(* IEC 61131-3 sources: MotionTestBenchMaster/Logical/00_AID/Libraries/Sidel_Libraries/ITC/TCP_COM, 5 files *)

(* ---- TCP_COM.typ ---- *)
(********************************************************************
 * COPYRIGHT --
 ********************************************************************
 * Package: TCP
 * File: TCP.typ
 * Author: Marco.Nicoli
 * Created: October 25, 2016 : Initial version
 *********************************************************************)

TYPE
	TCP_DataType : 	STRUCT
		Connection_OK : BOOL;
		Com_Status : UINT; (*(0=Connect OK;1=Not Enabled;2=Error Sending;3=Error Receiving;10=Connection Waiting)*)
		Recv_Buffer : ARRAY[0..20]OF USINT;
		Send_Buffer : ARRAY[0..20]OF USINT;
	END_STRUCT;
	TCP_Status_Type :
		(
		DISABLED,
		INITIALIZE_FB,
		INITIAL_PING,
		READ_LOCAL_IP,
		OPEN_TCP,
		CFG_SERVER,
		CFG_CLIENT,
		ESTABLISHED_CONNECTION_AS_SERVER,
		ESTABLISHED_CONNECTION_AS_CLIENT,
		CLOSE1,
		CLOSE2,
		RECONNECTION
		);
	TCP_SendRec_Type :
		(
		COMM_IDLE,
		SEND_DATA,
		RECEIVE_DATA,
		COMM_PING
		);
	Ping_Status_Type :
		(
		NO_EXECUTION,
		EXECUTION,
		SUCCESSFUL,
		NO_RESPONSE,
		ERROR_INTERNAL
		);
END_TYPE

(* ---- PING_Fun.st ---- *)
FUNCTION_BLOCK PING_Fun
	IF NOT enable THEN
		PING_OK 			:= FALSE;
		ERR_NO_RESPONSE 	:= FALSE;
		ERR_INTERNAL	 	:= FALSE;
		ERROR 				:= FALSE;
		Status 				:= NO_EXECUTION;
		RETURN;
	END_IF;
	Fb_IcmpPing.pHost	:= ADR(IP_Address);
	Fb_IcmpPing.timeout := 50;
	CASE Status OF
		NO_EXECUTION:
			Fb_IcmpPing.enable  := FALSE;
			readResponse 	:= FALSE;
			PachetSent		:= 0;
			PachetRecived	:= 0;
			PachetLoss		:= 0;
			IF enable THEN
				Status := EXECUTION;
			END_IF;

		EXECUTION:
			Fb_IcmpPing.enable  := TRUE;
			IF Fb_IcmpPing.status = ERR_FUB_BUSY THEN
				readResponse := TRUE;
			END_IF
			IF readResponse THEN
				CASE Fb_IcmpPing.status OF
					ERR_OK:
						PachetSent 		:= PachetSent +1;
						PachetRecived 	:= PachetRecived +1;

					icmpERR_NO_RESPONSE:
						PachetSent 		:= PachetSent +1;
						PachetLoss 		:= PachetLoss +1;

					ERR_FUB_BUSY,
					ERR_FUB_ENABLE_FALSE:

					icmpERR_PARAMETER,
					icmpERR_SOCKET_CREATE,
					icmpERR_SYSTEM:
						Status := ERROR_INTERNAL;
				END_CASE;
			END_IF
			IF PachetSent >= 4 THEN
				IF PachetLoss >= 1 THEN
					Status := NO_RESPONSE;
				ELSE
					Status := SUCCESSFUL;
				END_IF
			END_IF

		SUCCESSFUL, NO_RESPONSE, ERROR_INTERNAL:
			Fb_IcmpPing.enable  := FALSE;

	END_CASE;
	Fb_IcmpPing();

	PING_OK 			:= Status = SUCCESSFUL;
	ERR_NO_RESPONSE 	:= Status = NO_RESPONSE;
	ERR_INTERNAL	 	:= Status = ERROR_INTERNAL;
	ERROR 				:= ERR_NO_RESPONSE OR ERR_INTERNAL;
END_FUNCTION_BLOCK

(* ---- TCP_COM.fun ---- *)
(********************************************************************
 * COPYRIGHT --
 ********************************************************************
 * Package: TCP
 * File: TCP.typ
 * Author: Marco.Nicoli
 * Created: October 25, 2016 : Initial version
 *********************************************************************)

FUNCTION_BLOCK TCP_COM (*TCP communication function*)
	VAR_INPUT
		Enable_Com : BOOL; (*Enable Communication*)
		Enable_Server : BOOL; (*Enable the server mode (False = Client mode | True = Serve mode)*)
		ETH_Card : STRING[16] := 'IF2'; (*Optional Parameter
Work with the following syntax when using IF2 on board:
IF2
Work with the following syntax when using a POWERLINK card:
SL<x>.SS<y>.IF<z>.PLKETH or SL<x>.SS<y>.IF<z>.ETH
*)
		IP_Address : STRING[16]; (*Partner IP address. (e.g. '10.1.92.20') (as a string)*)
		Local_Port : UINT; (*Local port number.*)
		Remote_Port : UINT; (*Remote port number.*)
		Recv_Buffer : UDINT; (*Received data buffer address (string given as a pointer)*)
		Recv_Length : UDINT; (*Reiceved data maximum length (in bytes)*)
		Send_Buffer : UDINT; (*Data to send buffer address (string given as a pointer)*)
		Send_Length : UDINT; (*Sent data length (in bytes)*)
		Send_Time_Act : TIME; (*Data send time cadence (in ms) (typical value: 100ms)*)
		Rcv_Time_Out : TIME; (*Reception time out setpoint (in ms) (typical value: 1000ms)*)
	END_VAR
	VAR_OUTPUT
		Connection_OK : BOOL; (*True = both PLCs are connected*)
		PING_OK : BOOL;
		ERROR : BOOL;
		ERR_NO_RESPONSE : BOOL;
		ERR_INTERNAL : BOOL;
	END_VAR
	VAR
		WhoIsConnected : STRING[16]; (*Connected client IP address*)
		IP_AdressLocal : STRING[16];
		TON_SendTime : TON;
		TON_RcvTimeOut : TON;
		TON_TCP_EnDelay : TON;
		TON_ConnectionTimeOut : TON;
		ConnectionAttempt : UINT;
		fb_Ping : PING_Fun;
		fb_TcpOpen : TcpOpen; (*Communication opening function block*)
		fb_TcpServer : TcpServer; (*Server creation function block*)
		fb_TcpClient : TcpClient; (*Client function block*)
		fb_TcpSend : TcpSend; (*Data sending function block*)
		fb_TcpRecv : TcpRecv; (*Data receiving function block*)
		fb_TcpClose : TcpClose; (*Communication closing function block*)
		fb_CfgGetIPAddr : CfgGetIPAddr;
		oldTCP_Status : TCP_Status_Type;
		oldTCP_CommStatus : TCP_SendRec_Type;
		IP_LocalValid : BOOL;
		readResponse : BOOL;
		commResponse : BOOL;
		TCP_Status : TCP_Status_Type; (*Implemented communication block status*)
		TCP_CommStatus : TCP_SendRec_Type; (*Implemented communication block status*)
		TON_Connection_OK : TON;
	END_VAR
END_FUNCTION_BLOCK

FUNCTION_BLOCK PING_Fun (*TODO: Add your comment here*) (*$GROUP=User,$CAT=User,$GROUPICON=User.png,$CATICON=User.png*)
	VAR_INPUT
		enable : BOOL;
		IP_Address : STRING[80];
	END_VAR
	VAR_OUTPUT
		PING_OK : BOOL;
		ERROR : BOOL;
		ERR_NO_RESPONSE : BOOL;
		ERR_INTERNAL : BOOL;
	END_VAR
	VAR
		Status : Ping_Status_Type;
		Fb_IcmpPing : IcmpPing;
		PachetRecived : USINT;
		PachetSent : USINT;
		PachetLoss : USINT;
		readResponse : BOOL;
	END_VAR
END_FUNCTION_BLOCK

(* ---- TCP_Fun.st ---- *)
(********************************************************************
 * COPYRIGHT --
 ********************************************************************
 * Package: TCP
 * File: TCP.st
 * Author: Marco.Nicolì
 * Created: October 25, 2016 : Initial version
 * Modified: November 15, 2016 : Something
 ********************************************************************)

FUNCTION_BLOCK TCP_COM
	CASE TCP_Status OF
		DISABLED:
			ConnectionAttempt 	:= 0;
			PING_OK 			:= FALSE;
			ERR_INTERNAL		:= FALSE;
			ERR_NO_RESPONSE		:= FALSE;
			TON_TCP_EnDelay.IN 	:= Enable_Com;
			TON_TCP_EnDelay.PT 	:= t#2s;
			TON_TCP_EnDelay();
			IF TON_TCP_EnDelay.Q THEN
				TON_TCP_EnDelay(IN := FALSE);
				TCP_Status := INITIALIZE_FB;
			END_IF

		INITIALIZE_FB:
			fb_Ping.enable 		:= FALSE;
			fb_TcpOpen.enable	:= FALSE;
			fb_TcpServer.enable	:= FALSE;
			fb_TcpClient.enable	:= FALSE;
			fb_TcpSend.enable	:= FALSE;
			fb_TcpRecv.enable	:= FALSE;
			fb_TcpClose.enable	:= FALSE;
			fb_CfgGetIPAddr.enable := FALSE;
			fb_Ping();
			fb_TcpOpen();
			fb_TcpServer();
			fb_TcpClient();
			fb_TcpSend();
			fb_TcpRecv();
			fb_TcpClose();
			fb_CfgGetIPAddr();

			TON_TCP_EnDelay.IN 	:= TRUE;
			TON_TCP_EnDelay.PT 	:= t#100ms;
			TON_TCP_EnDelay();
			IF TON_TCP_EnDelay.Q THEN
				TON_TCP_EnDelay(IN := FALSE);
				TCP_Status := INITIAL_PING;
			END_IF

		INITIAL_PING:
			fb_Ping.enable 		:= TRUE;
			fb_Ping.IP_Address 	:= IP_Address;
			fb_Ping();
			IF NOT Enable_Com THEN
				TCP_Status 	:= DISABLED;
			ELSIF fb_Ping.PING_OK THEN
				PING_OK 	:= TRUE;
				IF ETH_Card = '' THEN
					TCP_Status 	:= OPEN_TCP;
				ELSE
					TCP_Status 	:= READ_LOCAL_IP;
				END_IF
			ELSIF fb_Ping.ERROR THEN
				ERR_NO_RESPONSE := fb_Ping.ERR_NO_RESPONSE;
				ERR_INTERNAL	:= fb_Ping.ERR_INTERNAL;
				TCP_Status 		:= RECONNECTION;
			END_IF

		READ_LOCAL_IP:
			fb_CfgGetIPAddr.enable 	:= TRUE;
			fb_CfgGetIPAddr.pDevice := ADR(ETH_Card);
			fb_CfgGetIPAddr.pIPAddr := ADR(IP_AdressLocal);
			fb_CfgGetIPAddr.Len 	:= SIZEOF(IP_AdressLocal);
			fb_CfgGetIPAddr();
			IF fb_CfgGetIPAddr.status = ERR_FUB_BUSY THEN
				readResponse := TRUE;
			END_IF
			IF readResponse THEN
				IF fb_CfgGetIPAddr.status = ERR_OK AND NOT (IP_AdressLocal = 'ERROR') THEN
					IP_LocalValid := TRUE;
					TCP_Status 		:= OPEN_TCP;
				ELSIF fb_CfgGetIPAddr.status <> ERR_FUB_BUSY OR (IP_AdressLocal = 'ERROR') THEN
					IP_LocalValid := FALSE;
					TCP_Status 		:= OPEN_TCP;
				END_IF
			END_IF

		OPEN_TCP:
			fb_TcpOpen.enable	:= TRUE;
			IF IP_LocalValid THEN
				fb_TcpOpen.pIfAddr 	:= ADR(IP_AdressLocal);
			ELSE
				fb_TcpOpen.pIfAddr 	:= 0;
			END_IF
			fb_TcpOpen.port 	:= Local_Port;
			fb_TcpOpen.options 	:= tcpOPT_REUSEADDR;
			fb_TcpOpen();
			IF fb_TcpOpen.status = ERR_FUB_BUSY THEN
				readResponse := TRUE;
			END_IF
			IF readResponse THEN
				IF fb_TcpOpen.status = ERR_OK THEN
					IF Enable_Server THEN
						TCP_Status := CFG_SERVER;
					ELSE
						TCP_Status := CFG_CLIENT;
					END_IF
				ELSIF fb_TcpOpen.status = tcpERR_SOCKET_BIND THEN
					ERR_NO_RESPONSE	:= FALSE;
					TCP_Status 		:= CLOSE2;
				END_IF
			END_IF
			IF NOT Enable_Com THEN
				TCP_Status 	:= CLOSE2;
			END_IF

		CFG_SERVER:
			fb_TcpServer.enable 	:= TRUE;
			fb_TcpServer.ident 		:= fb_TcpOpen.ident;
			fb_TcpServer.backlog 	:= 1;
			fb_TcpServer.pIpAddr 	:= ADR(WhoIsConnected);
			fb_TcpServer();
			TON_ConnectionTimeOut.IN := fb_TcpServer.status = ERR_FUB_BUSY;
			TON_ConnectionTimeOut.PT := t#20s;
			TON_ConnectionTimeOut();
			IF fb_TcpServer.status = ERR_FUB_BUSY THEN
				readResponse := TRUE;
			END_IF
			IF readResponse THEN
				IF fb_TcpServer.status = ERR_OK THEN
					TCP_Status 	:= ESTABLISHED_CONNECTION_AS_SERVER;
				ELSIF (fb_TcpServer.status <> ERR_FUB_BUSY) AND (fb_TcpServer.status <> ERR_OK) THEN
					TCP_Status 		:= CLOSE1;
					ERR_INTERNAL	:= TRUE;
				END_IF
			END_IF
//			IF NOT Enable_Com OR TON_ConnectionTimeOut.Q THEN
//				TCP_Status 	:= CLOSE2;
//			END_IF

		CFG_CLIENT:
			fb_TcpClient.enable 	:= TRUE;
			fb_TcpClient.ident 		:= fb_TcpOpen.ident;
			fb_TcpClient.portserv 	:= Remote_Port;
			fb_TcpClient.pServer 	:= ADR(IP_Address);
			fb_TcpClient();
			IF fb_TcpClient.status = ERR_FUB_BUSY THEN
				readResponse := TRUE;
			END_IF
			IF readResponse THEN
				IF fb_TcpClient.status = ERR_OK THEN
					TCP_Status 	:= ESTABLISHED_CONNECTION_AS_CLIENT;
				ELSIF (fb_TcpClient.status <> ERR_FUB_BUSY) AND (fb_TcpClient.status <> ERR_OK) THEN
					ERR_INTERNAL	:= TRUE;
					TCP_Status 		:= CLOSE1;
				END_IF
			END_IF
			IF NOT Enable_Com THEN
				TCP_Status 	:= CLOSE1;
			END_IF

		ESTABLISHED_CONNECTION_AS_SERVER:
			TON_SendTime.IN := (TCP_CommStatus = RECEIVE_DATA);
			TON_SendTime.PT := Send_Time_Act;
			TON_SendTime();

			CASE TCP_CommStatus OF
				COMM_IDLE:
					TCP_CommStatus	:= SEND_DATA;

				SEND_DATA:
					fb_TcpSend.enable 	:= TRUE;
					fb_TcpSend.ident 	:= fb_TcpServer.identclnt;
					fb_TcpSend.pData 	:= Send_Buffer;
					fb_TcpSend.datalen 	:= Send_Length;
					fb_TcpSend();

					IF fb_TcpSend.status = ERR_FUB_BUSY THEN
						commResponse := TRUE;
					END_IF

					IF commResponse THEN
						IF fb_TcpSend.status	= ERR_OK THEN
							TCP_CommStatus	:= RECEIVE_DATA;
						ELSIF fb_TcpSend.status	= tcpERR_NOT_CONNECTED OR fb_TcpSend.status	= tcpERR_SYSTEM THEN
							TON_RcvTimeOut.IN := TRUE;
						END_IF
					END_IF

					IF TON_RcvTimeOut.Q THEN
						TON_RcvTimeOut.IN	:= FALSE;
						TCP_CommStatus		:= COMM_PING;
					END_IF

				RECEIVE_DATA:
					fb_TcpRecv.enable 	:= TRUE;
					fb_TcpRecv.ident 	:= fb_TcpServer.identclnt;
					fb_TcpRecv.pData 	:= Recv_Buffer;
					fb_TcpRecv.datamax 	:= Recv_Length;
					fb_TcpRecv();

					IF commResponse THEN
						IF TON_SendTime.Q AND (fb_TcpRecv.status = ERR_OK OR fb_TcpRecv.status = tcpERR_NO_DATA) THEN
							TCP_CommStatus	:= SEND_DATA;
						ELSIF fb_TcpRecv.status	= tcpERR_NOT_CONNECTED OR fb_TcpRecv.status	= tcpERR_NO_DATA OR fb_TcpSend.status = tcpERR_SYSTEM THEN
							TON_RcvTimeOut.IN := TRUE;
						ELSIF NOT fb_TcpRecv.status = ERR_FUB_BUSY OR fb_TcpRecv.status = ERR_OK THEN
							TON_RcvTimeOut.IN := FALSE;
						END_IF
					END_IF

					IF fb_TcpRecv.status = ERR_FUB_BUSY THEN
						commResponse := TRUE;
					END_IF

					IF TON_RcvTimeOut.Q THEN
						TON_RcvTimeOut.IN	:= FALSE;
						TCP_CommStatus		:= COMM_PING;
					END_IF

				COMM_PING:
					fb_Ping.enable 		:= TRUE;
					fb_Ping.IP_Address 	:= IP_Address;
					fb_Ping();
					IF fb_Ping.PING_OK THEN
						PING_OK 		:=	TRUE;
						TCP_CommStatus	:= RECEIVE_DATA;
					ELSIF fb_Ping.ERROR THEN
						ERR_NO_RESPONSE := fb_Ping.ERR_NO_RESPONSE;
						ERR_INTERNAL	:= fb_Ping.ERR_INTERNAL;
						TCP_Status 		:= CLOSE1;
					END_IF

			END_CASE

			TON_RcvTimeOut.PT := Rcv_Time_Out;
			TON_RcvTimeOut();

			IF TON_RcvTimeOut.Q OR NOT Enable_Com THEN
				TCP_Status 		:= CLOSE1;
				ERR_NO_RESPONSE := TRUE;
			END_IF

		ESTABLISHED_CONNECTION_AS_CLIENT:
			TON_SendTime.IN := (TCP_CommStatus = RECEIVE_DATA);
			TON_SendTime.PT := Send_Time_Act;
			TON_SendTime();

			CASE TCP_CommStatus OF
				COMM_IDLE:
					TCP_CommStatus	:= SEND_DATA;

				SEND_DATA:
					fb_TcpSend.enable 	:= TRUE;
					fb_TcpSend.ident 	:= fb_TcpOpen.ident;
					fb_TcpSend.pData 	:= Send_Buffer;
					fb_TcpSend.datalen 	:= Send_Length;
					fb_TcpSend();

					IF fb_TcpSend.status = ERR_FUB_BUSY THEN
						commResponse := TRUE;
					END_IF

					IF commResponse THEN
						IF fb_TcpSend.status = ERR_OK THEN
							TCP_CommStatus	:= RECEIVE_DATA;
						ELSIF fb_TcpSend.status	= tcpERR_NOT_CONNECTED OR fb_TcpSend.status	= tcpERR_SYSTEM THEN
							TON_RcvTimeOut.IN := TRUE;
						END_IF
					END_IF

					IF TON_RcvTimeOut.Q THEN
						TON_RcvTimeOut.IN	:= FALSE;
						TCP_CommStatus		:= COMM_PING;
					END_IF

				RECEIVE_DATA:
					fb_TcpRecv.enable 	:= TRUE;
					fb_TcpRecv.ident 	:= fb_TcpOpen.ident;
					fb_TcpRecv.pData 	:= Recv_Buffer;
					fb_TcpRecv.datamax 	:= Recv_Length;
					fb_TcpRecv();

					IF commResponse THEN
						IF TON_SendTime.Q AND (fb_TcpRecv.status = ERR_OK OR fb_TcpRecv.status = tcpERR_NO_DATA) THEN
							TCP_CommStatus	:= SEND_DATA;
						ELSIF fb_TcpRecv.status	= tcpERR_NOT_CONNECTED OR fb_TcpRecv.status	= tcpERR_NO_DATA OR fb_TcpSend.status = tcpERR_SYSTEM THEN
							TON_RcvTimeOut.IN := TRUE;
						ELSIF NOT fb_TcpRecv.status = ERR_FUB_BUSY OR fb_TcpRecv.status = ERR_OK THEN
							TON_RcvTimeOut.IN := FALSE;
						END_IF
					END_IF

					IF fb_TcpRecv.status = ERR_FUB_BUSY THEN
						commResponse := TRUE;
					END_IF

					IF TON_RcvTimeOut.Q THEN
						TON_RcvTimeOut.IN	:= FALSE;
						TCP_CommStatus		:= COMM_PING;
					END_IF

				COMM_PING:
					fb_Ping.enable 		:= TRUE;
					fb_Ping.IP_Address 	:= IP_Address;
					fb_Ping();
					IF fb_Ping.PING_OK THEN
						PING_OK 		:=	TRUE;
						TCP_CommStatus	:= RECEIVE_DATA;
					ELSIF fb_Ping.ERROR THEN
						ERR_NO_RESPONSE := fb_Ping.ERR_NO_RESPONSE;
						ERR_INTERNAL	:= fb_Ping.ERR_INTERNAL;
						TCP_Status 		:= CLOSE1;
					END_IF

			END_CASE

			TON_RcvTimeOut.PT := Rcv_Time_Out;
			TON_RcvTimeOut();

			IF TON_RcvTimeOut.Q OR NOT Enable_Com THEN
				TCP_Status 		:= CLOSE1;
				ERR_NO_RESPONSE := TRUE;
			END_IF

		CLOSE1:
			IF Enable_Server THEN
				PING_OK := FALSE;
				fb_TcpClose.enable 	:= TRUE;
				fb_TcpClose.ident 	:= fb_TcpServer.identclnt;
				fb_TcpClose();
				IF fb_TcpClose.status = ERR_FUB_BUSY THEN
					readResponse := TRUE;
				END_IF
				IF readResponse THEN
					IF fb_TcpClose.status = ERR_OK OR fb_TcpClose.status = tcpERR_INVALID_IDENT THEN
						TCP_Status 	:= CLOSE2;
					END_IF
				END_IF
			ELSE
				TCP_Status 	:= CLOSE2;
			END_IF

		CLOSE2:
			PING_OK := FALSE;
			fb_TcpClose.enable 	:= TRUE;
			fb_TcpClose.ident 	:= fb_TcpOpen.ident;
			fb_TcpClose();
			IF fb_TcpClose.status = ERR_FUB_BUSY THEN
				readResponse := TRUE;
			END_IF
			IF readResponse THEN
				IF fb_TcpClose.status = ERR_OK OR fb_TcpClose.status = tcpERR_INVALID_IDENT THEN
					IF NOT Enable_Com THEN
						TCP_Status 	:= DISABLED;
					ELSE
						TCP_Status 	:= RECONNECTION;
					END_IF
				END_IF
			END_IF

		RECONNECTION:
			PING_OK := FALSE;
			TON_TCP_EnDelay.IN := TRUE;
			IF ConnectionAttempt = 0 THEN
				TON_TCP_EnDelay.PT := t#100ms;
			ELSIF ConnectionAttempt < 5 THEN
				TON_TCP_EnDelay.PT := t#5s;
			ELSIF ConnectionAttempt < 11 THEN
				TON_TCP_EnDelay.PT := t#30s;
			ELSIF ConnectionAttempt < 20 THEN
				TON_TCP_EnDelay.PT := t#5m;
			END_IF
			TON_TCP_EnDelay();
			IF TON_TCP_EnDelay.Q THEN
				TON_TCP_EnDelay(IN := FALSE);
				ConnectionAttempt := ConnectionAttempt + 1;
				TCP_Status := INITIALIZE_FB;
			ELSIF NOT Enable_Com THEN
				TCP_Status 	:= DISABLED;
			END_IF
	END_CASE

	IF TCP_Status <> oldTCP_Status THEN
		oldTCP_Status := TCP_Status;
		TON_ConnectionTimeOut(IN := FALSE);
		readResponse := FALSE;
	END_IF

	IF TCP_CommStatus <> oldTCP_CommStatus THEN
		oldTCP_CommStatus := TCP_CommStatus;
		commResponse := FALSE;
	END_IF

	TON_Connection_OK.IN := (TCP_Status = ESTABLISHED_CONNECTION_AS_SERVER) OR (TCP_Status = ESTABLISHED_CONNECTION_AS_CLIENT);
	TON_Connection_OK.PT := t#3s;
	TON_Connection_OK();
	Connection_OK := TON_Connection_OK.Q;

	IF Connection_OK THEN
		ConnectionAttempt 	:= 0;
		ERR_INTERNAL		:= FALSE;
		ERR_NO_RESPONSE		:= FALSE;
	END_IF

	ERROR := ERR_INTERNAL OR ERR_NO_RESPONSE;
END_FUNCTION_BLOCK

(* ---- TCP_COM.var ---- *)
(********************************************************************
 * COPYRIGHT --
 ********************************************************************
 * Library: TCP_COMM
 * File: TCP_COMM.var
 * Author: SIDEL Conveying France
 * Created: October 02, 2008
 ********************************************************************
 * Constants of library TCP_COM
 ********************************************************************)
VAR CONSTANT
	TCP_Connected_OK : USINT := 0;
	TCP_Error_Sending : USINT := 2;
	TCP_Connection_Waiting : USINT := 10;
	TCP_Error_Receiving : USINT := 3;
	TCP_Not_Enabled : UINT := 1;
END_VAR
